SUBAPPLICATION ButtonT_AE_AX (* 1 Button (Trigger) und GreenWhiteBackground, gebuendelt hinter einem einzigen AE_AX-Plug (bidirektional: Trigger raus, Zustand rein) - HMI-Teil, ohne jeden OPC-UA-Bezug, wiederverwendbar. Button-Pendant zu SoftKeyT_AE_AX. *)
  (* Standard: 61499-2; Description: Copyright (c) 2026 Meisterschulen am Ostbahnhof This program and the accompanying materials are made available under the terms of the Eclipse Public License 2.0 which is available at https://www.eclipse.org/legal/epl-2.0/ SPDX-License-Identifier: EPL-2.0 *)
  (* Version 1.0, 2026-09-12, Franz Höpfinger, Meisterschulen am Ostbahnhof, initial implementation - Button-Pendant zu SoftKeyT_AE_AX (Softkey_IE ersetzt durch Button_IE, SK_RELEASED durch BT_PRESSED_LATCHED). *)
  PACKAGE MyLib::sys;
  IMPORT isobus::UT::Q::const::IDs::ID_NULL;
  IMPORT isobus::UT::io::Button::ButtonActivationCode::BT_PRESSED_LATCHED;
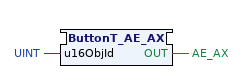
  VAR_INPUT
    u16ObjId : UINT := ID_NULL; (* Object ID Button/Background *)
  END_VAR
  PLUGS
    OUT : adapter::types::bidirectional::AE_AX; (* Trigger (out), Zustand (in) *)
  END_PLUGS
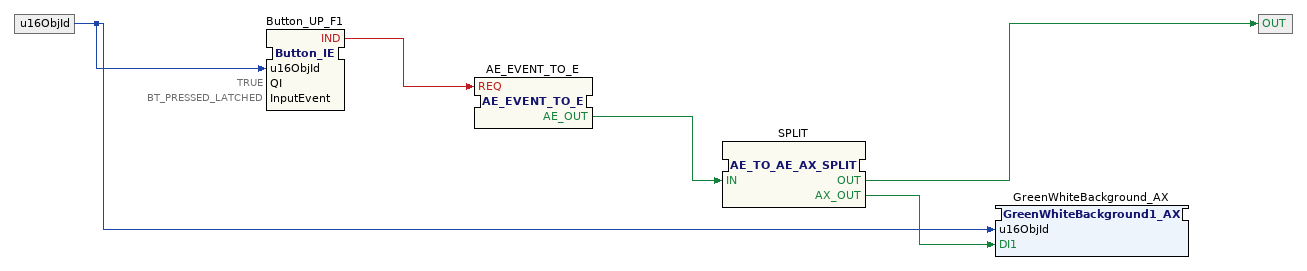
  FBS
    Button_UP_F1 : isobus::UT::io::Button::Button_IE(QI := TRUE, InputEvent := BT_PRESSED_LATCHED);
    AE_EVENT_TO_E : adapter::conversion::unidirectional::AE_EVENT_TO_E;
    SPLIT : adapter::events::bidirectional::AE_TO_AE_AX_SPLIT;
  END_FBS
  SUBAPPS
    GreenWhiteBackground_AX : MyLib::sys::GreenWhiteBackground1_AX;
  END_SUBAPPS
  EVENT_CONNECTIONS
    Button_UP_F1.IND TO AE_EVENT_TO_E.REQ;
  END_CONNECTIONS
  DATA_CONNECTIONS
    u16ObjId TO Button_UP_F1.u16ObjId;
    u16ObjId TO GreenWhiteBackground_AX.u16ObjId;
  END_CONNECTIONS
  ADAPTER_CONNECTIONS
    AE_EVENT_TO_E.AE_OUT TO SPLIT.IN;
    SPLIT.OUT TO OUT;
    SPLIT.AX_OUT TO GreenWhiteBackground_AX.DI1;
  END_CONNECTIONS
END_SUBAPPLICATION
